// TwinCAT 3 PLC project ActiveX_PLC
// ProgramVersion: 3.1.4023.0
// libraries:
//   Tc2_Standard, * (Beckhoff Automation GmbH)
//   Tc2_System, * (Beckhoff Automation GmbH)
//   Tc3_Module, * (Beckhoff Automation GmbH)
//   VisuSymbols,3.5.10.0,System
// project tree:
//   / GlobalTextList.TcGTLO, PlcTask.TcTTO, Visualization Manager.TcVMO (not stored)
//   POUs/ MAIN.TcPOU
//   VISUs/ Visualization.TcVIS
// real-time tasks:
//   TASK PlcTask: cycle T#10ms, priority 20, ADS port 350

CONFIGURATION ActiveX_PLC
    RESOURCE PLC ON TwinCAT3
        TASK PlcTask(INTERVAL := T#10ms, PRIORITY := 20);
        PROGRAM MAIN WITH PlcTask : MAIN;
    END_RESOURCE
END_CONFIGURATION

// ---- POUs/MAIN.TcPOU
PROGRAM MAIN
VAR
	bLoad 	: BOOL;
	sPath	: STRING := 'C:\Temp\TC3_SyncUnits.pdf';
END_VAR

END_PROGRAM

// ---- GlobalTextList.TcGTLO
TEXTLIST GlobalTextList
  287 = 'Load PDF'
  904 = 'Path: %s'
END_TEXTLIST

// ---- VISUs/Visualization.TcVIS
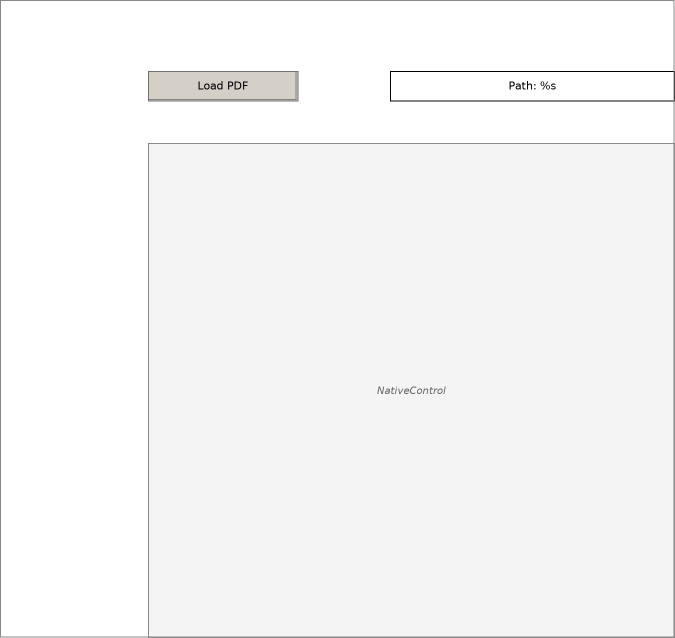
VISUALIZATION Visualization  // 675x638
    NativeControl (148,143 527x495)
        Calls[0]: Method=LoadFile, Variable=MAIN.bLoad
        Parameters[0]: Var=MAIN.sPath
        p3873840581: AcroPDF.PDF.1
    Button (148,71 150x30), "Load PDF"
        tap MAIN.bLoad
    Rectangle (390,71 285x30), "Path: %s", text variable: MAIN.sPath
END_VISUALIZATION
